// Function block for AC motors controlled with the LENZE d-31855 frequency inverter
FUNCTION_BLOCK FB_Component_ACmotor IMPLEMENTS I_Component
VAR_INPUT
	sName			: STRING[50];
	tTimeout		: TIME := T#0MS;
END_VAR

VAR_OUTPUT
	eJogFreq		: E_LenzeJogFreq := E_LenzeJogFreq.FOFF;
	
	bEnabled     	: BOOL;
	eState			: E_State := E_State.DISABLED;
	sStatusText 	: STRING[100];
END_VAR

VAR_IN_OUT
	bDeviceActive	: BOOL;	
	bE1jog1			: BOOL;					// jog func b1
	bE2jog2			: BOOL;					// jog func b2
	bE3DCbrake		: BOOL;					// DC injection brake
	eE4Direction	: BOOL;					// motor direction
END_VAR

VAR
	eLastState		: E_State;
	tTimeoutTimer	: TON;
END_VAR


VAR CONSTANT
	DISABLED		: E_State := E_State.DISABLED;
	READY			: E_State := E_State.READY;
	BUSY			: E_State := E_State.BUSY;
	DONE			: E_State := E_State.DONE;
	HALTED			: E_State := E_State.HALTED;
	TIMEOUT			: E_State := E_State.TIMEOUT;
	
	FOFF	: E_LenzeJogFreq := E_LenzeJogFreq.FOFF;
	F1		: E_LenzeJogFreq := E_LenzeJogFreq.F1;
	F2		: E_LenzeJogFreq := E_LenzeJogFreq.F2;
	F3		: E_LenzeJogFreq := E_LenzeJogFreq.F3;
END_VAR

tTimeoutTimer(PT := tTimeout);

CASE eState OF
	DISABLED:	sStatusText := '';
	
	READY:	 	sStatusText := 'Motor not moving, waiting for instruction';
				IF eJogFreq <> FOFF THEN
					eState := BUSY;
				END_IF
				
	BUSY: 		IF NOT bDeviceActive THEN
					sStatusText := 'frequency inverter not active';
				ELSE
					CASE eJogFreq OF
						FOFF: 	eState		:= E_State.TIMEOUT;		
						F1: 	sStatusText := CONCAT('motor running ', CONCAT(SEL(eE4Direction = TRUE, 'CCW','CW'), ' at freq 1'));		
						F2: 	sStatusText := CONCAT('motor running ', CONCAT(SEL(eE4Direction = TRUE, 'CCW','CW'), ' at freq 2'));				
						F3: 	sStatusText := CONCAT('motor running ', CONCAT(SEL(eE4Direction = TRUE, 'CCW','CW'), ' at freq 3')); 	
					END_CASE
				END_IF
	
	TIMEOUT: 	sStatusText := 'motor timeout';
				tTimeoutTimer(IN := TRUE);
				
				IF tTimeoutTimer.Q THEN
					eState := E_State.DONE;
				END_IF
				
	DONE: 		sStatusText := 'motor instruction done';
				bE1jog1 	:= FALSE;
				bE2jog2 	:= FALSE;
				M_Resume();
	
	HALTED: 	sStatusText := 'motor halted';
				bE1jog1		:= FALSE;
				bE2jog2		:= FALSE;

END_CASE

METHOD M_Disable : BOOL
VAR_INPUT
END_VAR
IF eState = DONE OR eState = READY THEN
	bEnabled	:= FALSE;
	eState		:= DISABLED;
END_IF
END_METHOD

METHOD M_Enable : BOOL
VAR_INPUT
END_VAR
IF eState = DISABLED THEN
	bEnabled	:= TRUE;
	eState 		:= READY;
END_IF
END_METHOD

METHOD M_Halt : BOOL
VAR_INPUT
END_VAR
eLastState 	:= eState;
eState 		:= HALTED;
END_METHOD

METHOD M_Reset : BOOL
VAR_INPUT
END_VAR
// has no use here
END_METHOD

METHOD M_Resume : BOOL
VAR_INPUT
END_VAR
CASE eState OF
	HALTED	: eState := eLastState;
	DONE	: eState := READY;
END_CASE
END_METHOD

METHOD M_SetDir : BOOL
VAR_INPUT
	Direction: E_RotationDirection;
END_VAR
eE4Direction := TO_BOOL(Direction);
END_METHOD

METHOD M_SetFreq : BOOL
VAR_INPUT
	Frequency: E_LenzeJogFreq;
END_VAR
eJogFreq := Frequency;

IF bDeviceActive THEN
	CASE eJogFreq OF
		FOFF: 	bE1jog1 	:= FALSE;
				bE2jog2 	:= FALSE;
				
		F1: 	bE1jog1 	:= TRUE;
				bE2jog2 	:= FALSE;
				
		F2: 	bE1jog1 	:= TRUE;
				bE2jog2 	:= TRUE;

		F3: 	bE1jog1 	:= FALSE;
				bE2jog2 	:= TRUE;
	END_CASE
END_IF
END_METHOD

METHOD M_Stop : BOOL
VAR_INPUT
END_VAR
IF eState <> BUSY OR eState <> HALTED OR eState <> TIMEOUT THEN
	eState := DONE;
END_IF
END_METHOD

END_FUNCTION_BLOCK

(* stored: Version 1.1.0.1, ProductVersion 3.1.4024.15
   POU FB_Component_ACmotor: Id {4bee0a47-7e8d-4a20-bf36-74643afc4427}, SpecialFunc None
   Method M_Disable: Id {71c72c1b-90db-4155-81a4-5bff4fcce209}
   Method M_Enable: Id {c92aa9f1-9d9c-44c7-a5b6-0e765f9c3f9f}
   Method M_Halt: Id {53708385-0949-4c5c-b3ef-98a2fb526cc6}
   Method M_Reset: Id {5a44a633-eb63-43a4-a451-a200476d7f2f}
   Method M_Resume: Id {66616ade-f252-442d-bf57-ed976b2ae351}
   Method M_SetDir: Id {d6a197ac-aaf3-4f2e-919c-b2334f169d78}
   Method M_SetFreq: Id {387ee47f-c4da-4cf1-a6b6-e28ea3f37257}
   Method M_Stop: Id {88cf4fbd-bea8-4d67-8643-88a00f690975} *)
